// TIA Portal V20 export
DATA_BLOCK "Temp_Sig"   // DB408
// stored: Access Published, MemoryReserve 100, Namespace Unit1
   VAR
      AlwaysOff : Bool;
      Bypass : Bool;
   END_VAR
BEGIN
END_DATA_BLOCK
